# EPICS SNL sequencer program: scanApp/src/xena_sncscan_new.stt
//#################################################
//# ###                                       ### #
//# ### Epics SNL Routines for		      ### #
//# ### Scan System	                      ### #
//# ###                                       ### #
//# ### author: D. Hampai - M. Montis         ### #
//# ###                                       ### #
//# ### Ref 1.0; 2025-12-04                   ### #
//#################################################
//#
//
program xena_sncscan

%{
#include <math.h>
#include <stdlib.h>

#define MAX_MOTORS 20

}%

/*=================== Declarations =========================*/

option +r;       /* Make the generated code reentrant, thus allowing more than one instance of the program to run on an IOC */
//
string name_exp_pv;
assign name_exp_pv to "{user}:experiment";
monitor name_exp_pv;
//
string name_exp[40];
//
// General Scan Configuration
//
int status_mode;
assign status_mode to "{user}:status";
monitor status_mode;
string actual_status;
assign actual_status to "{user}:state";
monitor actual_status;

int scan_busy;
assign scan_busy to "{user}:scan_busy";
monitor scan_busy;
int scan_pause;
assign scan_pause to "{user}:scan_pause";
monitor scan_pause;
int scan_restart;
assign scan_restart to "{user}:scan_restart";
monitor scan_restart;
int scan_abort;
assign scan_abort to "{user}:scan_abort";
monitor scan_abort;

int end_scan;

//
//	Definition Scan Parameters
//
int num_mot;
assign num_mot to "{user}:num_motor";
monitor num_mot;
int num_det;
assign num_det to "{user}:num_detector";
monitor num_det;

double start[20];
assign start to "{user}:start";
monitor start;
double end[20];
assign end to "{user}:end";
monitor end;
double step[20];
assign step to "{user}:step";
monitor step;
//
double posit[20];
int index[20];
int npoints[20];
//
int total_points;
assign total_points to "{user}:total_points";
monitor total_points;
int current_point;
assign current_point to "{user}:current_point";
monitor current_point;
double scan_progress;
assign scan_progress to "{user}:scan_progress";
monitor scan_progress;
//
//	Definition Loop Parameters
//
int flags[20];
//
//	Definition Motors Variables
//
string motor[20];
assign motor to "{user}:motor";
monitor motor;

string mot_command[6];
assign mot_command to "{user}:motor_command";
monitor mot_command;
//
// Definition Detectors Variables
//
string detector[20];
assign detector to "{user}:detector";
monitor detector;

string det_command[6];
assign det_command to "{user}:detector_command";
monitor det_command;

// Local Strings
double motget;
assign motget to "";
monitor motget;
double motset;
assign motset to "";
monitor motset;

double detget;
assign detget to "";
monitor detget;
double detset;
assign detset to "";
monitor detset;

double pos;
double mov_wait;
double acq_wait;
//
//	Local Variables
//
double motor_mr[20];
assign motor_mr to {};
monitor motor_mr;
double motor_ma[20];
assign motor_ma to {};
monitor motor_ma;
int motor_reqmov[20];
assign motor_reqmov to {};
monitor motor_reqmov;
int motor_mov[20];
assign motor_mov to {};
monitor motor_mov;
int motor_reqpos[20];
assign motor_reqpos to {};
monitor motor_reqpos;
double motor_pos[20];
assign motor_pos to {};
monitor motor_pos;
//
int detector_reqstart[20];
assign detector_reqstart to {};
monitor detector_reqstart;
int detector_reqready[20];
assign detector_reqready to {};
monitor detector_reqready;
int detector_ready[20];
assign detector_ready to {};
monitor detector_ready;
int detector_reqdata[20];
assign detector_reqdata to {};
monitor detector_reqdata;
double detector_data[20];
assign detector_data to {};
monitor detector_data;
int detector_type[20];
assign detector_type to{};
monitor detector_type;
//

int i;
int j;
int k;
int command;
char temp_string[80];
char temp_status[80];
//
//
//
//
ss scan_status_mode {
/*=================== Start Program =========================*/
        state init {
                when (status_mode==0) {
			pvGet(name_exp_pv,SYNC);
//			printf("the experiment is %s\n", name_exp_pv);
//			pvAssign(name_exp,name_exp_pv);
//			printf("the experiment is %s\n", name_exp);
//
                        printf("\n **********************\n");
                        printf("\n *** Ready for Scan ***\n");
                        printf("\n ***    Exp Xena    ***\n");
                        printf("\n **********************\n");
			strcpy(actual_status, "Starting Scan Program");
			pvPut(actual_status,SYNC);
			} state idle
        }
	state idle {
		when (status_mode==1) {
                        printf("\n ********************\n");
                        printf("\n *** Assign Motor ***\n");
                        printf("\n ********************\n");
		} state assign_motor
		when (status_mode==2) {
                        printf("\n ***********************\n");
                        printf("\n *** Assign Detector ***\n");
                        printf("\n ***********************\n");
		} state assign_detector
		when (status_mode==3) {
                        printf("\n ***************************\n");
                        printf("\n *** Initialization Loop ***\n");
                        printf("\n ***************************\n");
                } state init_loop
                when (status_mode==4) {
                        printf("\n ********************\n");
                        printf("\n *** Prepare Loop ***\n");
                        printf("\n ********************\n");
		} state prepare_loop
                when (status_mode==5) {
                        printf("\n ******************\n");
                        printf("\n *** Inner Loop ***\n");
                        printf("\n ******************\n");
                } state inner_loop
                when (status_mode==6) {
                        printf("\n ******************\n");
                        printf("\n *** Dummy Loop ***\n");
                        printf("\n ******************\n");
                } state dummy_loop
	}
//        state idle {
/*=================== Assign Motor Varibles =========================*/
/*======================= status_mode = 1 ===========================*/
        state assign_motor {
//		when (status_mode==1) {
		when () {
			printf("num_mot = %d\n", num_mot);
			for (i = 0; i < num_mot; i++) {
				printf("index = %d\n", i);
//
				command=0;
				sprintf(temp_string, "%s:%s", motor[i], mot_command[command]);
				printf("%s\n", temp_string);
				pvAssign(motor_mr[i],temp_string);
//
                                command=1;
                                sprintf(temp_string, "%s:%s", motor[i], mot_command[command]);
                                printf("%s\n", temp_string);
                                pvAssign(motor_ma[i],temp_string);
//
                                command=2;
                                sprintf(temp_string, "%s:%s", motor[i], mot_command[command]);
                                printf("%s\n", temp_string);
                                pvAssign(motor_reqmov[i],temp_string);
//
                                command=3;
                                sprintf(temp_string, "%s:%s", motor[i], mot_command[command]);
                                printf("%s\n", temp_string);
                                pvAssign(motor_mov[i],temp_string);
//
                                command=4;
                                sprintf(temp_string, "%s:%s", motor[i], mot_command[command]);
                                printf("%s\n", temp_string);
                                pvAssign(motor_reqpos[i],temp_string);
//
                                command=5;
                                sprintf(temp_string, "%s:%s", motor[i], mot_command[command]);
                                printf("%s\n", temp_string);
                                pvAssign(motor_pos[i],temp_string);
			}
                        strcpy(actual_status, "Motors Parameters Assigned - Status 1");
                        pvPut(actual_status,SYNC);
			status_mode=0;
			pvPut(status_mode);
		} state idle
	}
/*=================== Assign Detector Varibles =========================*/
/*======================== status_mode = 2 =============================*/
        state assign_detector {
//                when (status_mode==2) {
                when () {
                        printf("num_det = %d\n", num_det);
                        for (i = 0; i < num_det; i++) {
                                printf("index = %d\n", i);
//
                                command=0;
                                sprintf(temp_string, "%s:%s", detector[i], det_command[command]);
                                printf("%s\n", temp_string);
                                pvAssign(detector_reqstart[i],temp_string);
//
                                command=1;
                                sprintf(temp_string, "%s:%s", detector[i], det_command[command]);
                                printf("%s\n", temp_string);
                                pvAssign(detector_reqdata[i],temp_string);
//
                                command=2;
                                sprintf(temp_string, "%s:%s", detector[i], det_command[command]);
                                printf("%s\n", temp_string);
                                pvAssign(detector_data[i],temp_string);
//
                                command=3;
                                sprintf(temp_string, "%s:%s", detector[i], det_command[command]);
                                printf("%s\n", temp_string);
                                pvAssign(detector_reqready[i],temp_string);
//
                                command=4;
                                sprintf(temp_string, "%s:%s", detector[i], det_command[command]);
                                printf("%s\n", temp_string);
                                pvAssign(detector_ready[i],temp_string);
//
                                command=5;
                                sprintf(temp_string, "%s:%s", detector[i], det_command[command]);
                                printf("%s\n", temp_string);
                                pvAssign(detector_type[i],temp_string);
                        }
                        strcpy(actual_status, "Detect. Parameters Assigned - Status 2");
                        pvPut(actual_status,SYNC);
                        status_mode=0;
                        pvPut(status_mode);
                } state idle
	}
/*=================== Initialize Loop =========================*/
/*=================== status_mode = 3 =========================*/

        state init_loop {
                when() {
			end_scan=0; // initialize end scan
			total_points = 1;
                        for (i = 0; i < num_mot; i++) {
                                flags[i]=0;  // init flags
                                posit[i]=start[i];
                                index[i]=0;
                                npoints[i] = ( (end[i]-start[i]) / step[i] ) + 1;
                                printf("the number steps fo %d motor is %d\n", i, npoints[i]);
				total_points *= npoints[i];
				printf("the step number is %d\n", total_points);
                        }
			pvPut(total_points,SYNC);
			current_point=0;
			pvPut(current_point,SYNC);
			scan_busy=0;
                        pvPut(scan_busy,SYNC);
                        scan_restart=0;
			pvPut(scan_restart,SYNC);
                        scan_pause=0;
                        pvPut(scan_pause,SYNC);
                        scan_abort=0;
                        pvPut(scan_abort,SYNC);
//
                        strcpy(actual_status, "Scan Initialized - Status 3");
                        pvPut(actual_status,SYNC);
                        status_mode=0;
                        pvPut(status_mode);
                } state idle
        }

/*=================== Preparing Scan =========================*/
/*=================== status_mode = 4 ========================*/
        state prepare_loop {
//		when (status_mode==3) {
		when () {
			printf("\n **************************\n");
			printf("\n *** Preparing for Scan ***\n");
			printf("\n **************************\n");
			for (i = 0; i < num_mot; i++) {
//				printf("motor to move = %d\n", i);
				motor_ma[i]=start[i];
				pvPut(motor_ma[i],SYNC);
				motor_reqmov[i]=1;
//				printf("request moving = %d\n", motor_reqmov[i]);
					printf("1");
                                pvPut(motor_reqmov[i],SYNC);
					printf("2");
                                pvGet(motor_mov[i],SYNC);
					printf("3");
				printf("status moving = %d\n", motor_mov[i]);
				while(motor_mov[i]<1) {
					motor_reqmov[i]=1;
//					printf("request moving = %d\n", motor_reqmov[i]);
					pvPut(motor_reqmov[i],SYNC);
					pvGet(motor_mov[i],SYNC);
//					printf("status moving = %d\n", motor_mov[i]);
				}
				pvGet(motor_pos[i], SYNC);
//				printf("Position = %f\n", motor_pos[i]);
			}
			flags[0]=1; // Necessary to start the run
                        strcpy(actual_status, "Ready to Start");
                        pvPut(actual_status,SYNC);
                        status_mode=0;
                        pvPut(status_mode);
		} state dummy_loop
	}
/*=================== Inner Loop =========================*/
/*================= status_mode = 5 ======================*/
        state inner_loop {
//		when (status_mode==4) {
		when () {
			for (i=0; i < num_mot; i++) {
				posit[i]=start[i];
			}
//
                        printf("\n *************************\n");
                        printf("\n ***** Starting Scan *****\n");
                        printf("\n *************************\n");
                        strcpy(actual_status, "Starting Scan... %s is busy!!!");
                        pvPut(actual_status,SYNC);
//
			while (posit[num_det-1]>end[num_det-1]) {
				for (j=0; j < num_det; j++) {
					detector_reqstart[j]=1;
					pvPut(detector_reqstart[j],SYNC);
					printf("Starting Acquisition");
					detector_reqready[j]=1;
					pvPut(detector_reqready[j],SYNC);
					pvGet(detector_ready[j],SYNC);
					while(detector_ready[j]<1) {
						detector_reqready[j]=1;
						pvPut(detector_reqready[j],SYNC);
						pvGet(detector_ready[j],SYNC);
					}
					detector_reqdata[j]=1;
					pvPut(detector_reqdata[j],SYNC);
					pvGet(detector_data[j],SYNC);
					printf("The result for Detector %d = %f", j, detector_data[j]);
				}
			}
//
//
//
                        strcpy(actual_status, "Scan Finished");
                        pvPut(actual_status,SYNC);
                        status_mode=0;
                        pvPut(status_mode);
		} state idle
	}

/*=================== Dummy Loop =========================*/
/*================= status_mode = 6 ======================*/
// DEVO FARE UNA SERIE DI LOOP PER DIVERSI MOTORI
        state dummy_loop {
		when(scan_abort==1) {
			printf("Scan Aborted by User\n");
		} state abort_scan
//
		when() {
                        printf("\n *******************************\n");
                        printf("\n ***** Starting Dummy Scan *****\n");
                        printf("\n *******************************\n");
//

			snprintf(temp_status, sizeof(temp_status), "Starting Scan... %s is busy!!!", name_exp_pv);
//                        strcpy(actual_status, "Starting Scan... %s is busy!!!", name_exp_pv);
                        strcpy(actual_status, temp_status);
                        pvPut(actual_status,SYNC);
                        status_mode=0;
                        pvPut(status_mode);
		} state loops
	}

// LOOP Acquisizione
	state loops {
		when() {
		} state acquiring
	}

// LOOP NUOVE POSIZIONI
        state positions {
                when() {
			for (i=0; i<num_mot; i++) {
				if (flags[i] == 1) {
					if (index[i]==npoints[i]-1) {
						flags[i]=2;
						posit[i]=start[i];
						index[i]=0;
					} else {
						posit[i]=step[i]+posit[i];
						index[i]=index[i]+1;
					}
					if (flags[i] == 2 && i == num_mot-1) {
                                                end_scan=1;
					} else if (flags[i] == 2) {
						flags[i+1]=1;
					} else {
//						printf
					}
				}
			}
		} state moving
	}

// LOOP MOVIMENTO MOTORI
	state moving {
                when(scan_abort==1) {
                        printf("Scan Aborted by User\n");
                } state abort_scan
                when(scan_pause==1) {
                        printf("Scan Aborted by User\n");
                } state pause_scan
		when() {
                        for (i = 0; i < num_mot; i++) {
                                motor_ma[i]=posit[i];
                                pvPut(motor_ma[i],SYNC);
                                motor_reqmov[i]=1;
                                pvPut(motor_reqmov[i],SYNC);
                                pvGet(motor_mov[i],SYNC);
	                        while(motor_mov[i]<1) {
                                        motor_reqmov[i]=1;
                                        pvPut(motor_reqmov[i],SYNC);
                                        pvGet(motor_mov[i],SYNC);
                                }
                                pvGet(motor_pos[i], SYNC);
                        }
//
//			Reset Flags
//
			for(i=0; i<num_mot; i++) {
				flags[i]=0;
			}
			flags[0]=1;
//
                        status_mode=0;
                        pvPut(status_mode);
		} state loops
	}

// LOOP ACQUISIZIONI
//	EXIT
	state acquiring {
		when (end_scan==1) {
		} state ending
//	Doing Acquisition
		when () {
			for (j=0; j < num_det; j++) {
				detector_reqstart[j]=1;
				pvPut(detector_reqstart[j],SYNC);
				printf("Starting Acquisition");
				detector_reqready[j]=1;
				pvPut(detector_reqready[j],SYNC);
				pvGet(detector_ready[j],SYNC);
				while(detector_ready[j]<1) {
					detector_reqready[j]=1;
					pvPut(detector_reqready[j],SYNC);
					pvGet(detector_ready[j],SYNC);
				}
				detector_reqdata[j]=1;
				pvPut(detector_reqdata[j],SYNC);
				pvGet(detector_data[j],SYNC);
				printf("The result for Detector %d = %f", j, detector_data[j]);
			}
//
			printf("%d, %f, %f\n",current_point,posit[0],posit[1]);
			printf("%d, %f, %f\n",current_point,motor_pos[0],motor_pos[1]);
			current_point++;
		} state positions

	}

// END SCAN
	state ending {
                when() {
                        printf("\n ****************\n");
                        printf("\n *** End Scan ***\n");
                        printf("\n ****************\n");
                        status_mode=0;
                        pvPut(status_mode,SYNC);
                } state idle
	}

/*=================== Abort Scan =========================*/
	state abort_scan {
		when () {
			printf("rasterScan: Cleaning up after abort\n");
//			scan_running = 0;
//			pvPut(scan_running);
			scan_progress = 0;
			pvPut(scan_progress,SYNC);
			scan_abort = 0;
			pvPut(scan_abort,SYNC);
			status_mode=0;
			pvPut(status_mode,SYNC);
		} state idle
	}
/*=================== Pause =========================*/
	state pause_scan {
                when(scan_abort==1) {
                        printf("Scan Aborted by User\n");
                } state abort_scan
//
		when (scan_restart==1) {
                        scan_pause = 0;
                        pvPut(scan_pause,SYNC);
		} state moving
		when () {
			pvGet(scan_restart,SYNC);
			epicsThreadSleep(0.5);
		} state pause_scan
	}
}

/*
SPDX-FileCopyrightText: 1998 Argonne National Laboratory

SPDX-License-Identifier: EPICS
*/
